FUNCTION_BLOCK FB_EA_Interface
VAR_INPUT
	//Device Specifications - From Datasheet of the PSU/Load
	rMax_Current					: REAL;							
	rMax_Voltage					: REAL;
	rMax_Power						: REAL;
	rMax_Resistance					: REAL;
	
	//Setpoint
	rCurrent_Setpoint				: REAL;
	rVoltage_Setpoint				: REAL;
	rPower_Setpoint					: REAL;
	rResistance_Setpoint			: REAL;
	
	bRemote							: BOOL 		:= TRUE;
	bPowerStage						: BOOL;
END_VAR
VAR_OUTPUT
	bRemoteStatus					: BOOL;
	bPowerStageStatus				: BOOL;
	
	rCurrent_Actual					: REAL;
	rVoltage_Actual					: REAL;	
END_VAR
VAR
	stHWVar							: ST_EA_IO;
	                				
	eState							: (INIT, AUTO_ON, REMOTE, IDLE, POWER_STAGE_ON, POWER_STAGE_OFF, DONE, ERROR);  
	eParam							: (AUTO_ON,POWER_ON,REMOTE,POWER_STAGE);
	
	fbWriteCoe						: FB_ECCoeSdoWriteEx;
	
	nCoEVal							: ARRAY [1..4] OF UINT;
	bAutoOn							: BOOL;
	
END_VAR

VAR CONSTANT
	//CoE Index
	
	nCoeIdx_Remote					: WORD		:= 16#2193;
	nCoeIdx_AutoOn					: WORD		:= 16#2198;
	nCoeIdx_PowerOn					: WORD		:= 16#2199;
	nCoeIdx_PowerStage				: WORD		:= 16#2196;
		
END_VAR


ACT_Scaling();

CASE eState OF
	
	INIT: 
	
		fbWriteCoe(
			bExecute				:= FALSE);
			
				
		nCoEVal[AUTO_ON]			:= 65280;
		nCoEVal[POWER_ON]			:= 65535;
		nCoEVal[REMOTE]				:= 65280;
		nCoEVal[POWER_STAGE]		:= 0;
		
		IF NOT fbWriteCoe.bBusy
		AND stHWVar.stInfoData.nState=8						//Device in OP
		THEN
		
			eState					:= AUTO_ON;
			
		END_IF
					
			
	AUTO_ON:
	
		IF NOT fbWriteCoe.bBusy
		THEN
			ACT_AutoOn();
		ELSE
			eState					:= POWER_ON;
		END_IF
	
		
	
		
END_CASE

ACTION ACT_Auto_On:

END_ACTION

ACTION ACT_AutoOn:


fbWriteCoe(
	sNetID			:= stHWVar.stInfoData.stAdsAddr.netID,
	nSlaveAddr		:= stHWVar.stInfoData.stAdsAddr.port,
	nIndex			:= nCoeIdx_AutoOn,
	pSrcBuf			:= ADR(nCoEVal[AUTO_ON]),
	cbBufLen		:= SIZEOF(nCoeVal[AUTO_ON]),
	bExecute		:= TRUE);
END_ACTION

ACTION ACT_Scaling:


//Setpoint Scaling

stHWVar.stTxPDO.nCurrentSel			:= REAL_TO_UINT(rCurrent_Setpoint 	* (rMax_Current/65535));
stHWVar.stTxPDO.nPowerSel			:= REAL_TO_UINT(rPower_Setpoint 	* (rMax_Power/65535));
stHWVar.stTxPDO.nVoltageSel			:= REAL_TO_UINT(rVoltage_Setpoint 	* (rMax_Voltage/65535));
stHWVar.stTxPDO.nResistanceSel		:= REAL_TO_UINT(rResistance_Setpoint* (rMax_Resistance/65535));

//Actual Value Scaling


rCurrent_Actual						:= stHWVar.stRxPDO.nCurrentMon	/ rMax_Current;
rVoltage_Actual						:= stHWVar.stRxPDO.nVoltageMon	/ rMax_Voltage;
END_ACTION

END_FUNCTION_BLOCK

(* stored: Version 1.1.0.1, ProductVersion 3.1.4024.9
   POU FB_EA_Interface: Id {ef28b490-193f-413d-a266-c141ee8eb9a9}, SpecialFunc None
   Action ACT_Auto_On: Id {5a83d868-5e5e-424b-8253-995a6d9babe9}
   Action ACT_AutoOn: Id {5b2f47d3-0933-4a61-b98f-ae913c6e4fda}
   Action ACT_Scaling: Id {908518fa-127d-474d-b7dd-bb41556b928c} *)
